(* IEC 61131-3 sources: rules_plc/examples/library_deps_stubs, 4 files *)

(* ---- link_types.st ---- *)
(* Shared TYPE library at the bottom of a three-level dep chain.
Both eth and net take a `link_handle` by VAR_IN_OUT, so every library
downstream in the chain must see this struct definition -- exercising
rules_plc's relative-path `dependencies.plc.h` include chain. *)
TYPE

    link_handle:
STRUCT
    id: DINT := 0;
    state: DINT := 0;
END_STRUCT;

END_TYPE

(* ---- eth.st ---- *)
(* Middle-of-chain library: depends on link_types, so its generated
`dependencies.plc.h` re-exports link_types' headers by relative path. Every
FB here is `{external}` -- no ST implementation, so the C-level symbols
are supplied by whatever links against this library. *)

{external}
FUNCTION_BLOCK eth_status
    VAR_IN_OUT
        link: link_handle;
    END_VAR
    VAR_OUTPUT
        connected: BOOL := FALSE;
        speed_mbps: DINT := 0;
    END_VAR
END_FUNCTION_BLOCK

{external}
FUNCTION_BLOCK eth_reset
    VAR_IN_OUT
        link: link_handle;
    END_VAR
    VAR_OUTPUT
        done: BOOL := FALSE;
    END_VAR
END_FUNCTION_BLOCK

(* ---- net.st ---- *)
(* Top-of-chain library: depends on eth, which depends on link_types.
Its own generated `dependencies.plc.h` re-exports eth's headers by
relative path, and eth's `dependencies.plc.h` in turn re-exports
link_types' headers -- so the `link_handle` type used by-value in
net_send's VAR_IN_OUT resolves along the transitive chain. *)

{external}
FUNCTION_BLOCK net_send
    VAR_IN_OUT
        link: link_handle;
    END_VAR
    VAR_INPUT
        payload: DINT := 0;
    END_VAR
    VAR_OUTPUT
        ok: BOOL := FALSE;
    END_VAR
END_FUNCTION_BLOCK

(* ---- app_bin.st ---- *)
PROGRAM app_bin
    VAR
        my_link: link_handle;
        eth_st: eth_status;
        sender: net_send;
    END_VAR

    eth_st(link := my_link);
    IF eth_st.connected THEN
        sender(link := my_link, payload := 42);
    END_IF;
END_PROGRAM
